// Something with per-scan work.

//

// The bottom of the stack, with IQueryInterface beneath it. Every interface in

// this library reaches IQueryInterface through its own root, so any reference can

// be queried for any other role it plays.
INTERFACE I_TestCyclic EXTENDS __SYSTEM.IQueryInterface

// Called every scan, unconditionally, by whatever owns this object.

//

// The name is the contract. An Execute input would mean a trigger; an Enable

// input would mean held-while-wanted; CyclicLogic means there is no gating

// condition and the caller must not invent one.
METHOD CyclicLogic
END_METHOD

END_INTERFACE

(* stored: Version 1.1.0.1, ProductVersion 3.1.4026.18
   Itf I_TestCyclic: Id {7a95b8cb-aa86-4365-bddf-61d9232bfe04}
   Method CyclicLogic: Id {c46bd092-f06b-4fa1-937e-776ebadabca9} *)
